{attribute 'no_explicit_call' := 'do not call this function block directly'} 
FUNCTION_BLOCK ListOfReferences EXTENDS GenericList
VAR
	_ClassName : STRING := __POUNAME();
END_VAR

{attribute 'monitoring' := 'call'}
PROPERTY ClassName : STRING
GET
ClassName := _ClassName;
END_GET
END_PROPERTY

METHOD FB_init : BOOL
VAR_INPUT
	(* if TRUE, the retain variables are initialized (warm start / cold start)*)
	bInitRetains	: BOOL;
	(* if TRUE, the instance afterwards gets moved into the copy code (online change)*)
	bInCopyCode	: BOOL;
END_VAR
StoredTypeCategory := TYPE_CATEGORY.REFERENCE_TYPE;
END_METHOD

END_FUNCTION_BLOCK

(* stored: Version 1.1.0.1
   POU ListOfReferences: Id {9295f20c-0393-4907-879d-60a81a2ecb79}, SpecialFunc None
   Property ClassName: Id {60a3b590-daac-4d70-9d52-67e93feb03af}
   Get Get: Id {b60e12e2-b176-42e0-9b66-684a0cfc5a78}
   Method FB_init: Id {774629c4-adc8-4837-8ad3-5acb6900f79d} *)
